PROGRAM FB_RetourEfficace
VAR_INPUT
Ir_PosX : BOOL ;
Ir_PosY : BOOL ;	
Ir_PosXVoulue : BOOL ;	
Ir_PosYVoulue : BOOL ;	
END_VAR
VAR_OUTPUT
	
END_VAR
VAR
END_VAR

IF Ir_PosX

END_PROGRAM

(* stored: Version 1.1.0.1
   POU FB_RetourEfficace: Id {c14c33d8-dbee-4249-b7b2-87313a39a468}, SpecialFunc None *)
